(* CODESYS project Door.xml

Project tree, tasks and I/O mapping:
  function block Door [LD]
*)

// Door
FUNCTION_BLOCK Door
// The Door function block monitors the conditions required for locking and unlocking the door.
// The door should remained locked until a bag of ice is ready to be vended.
VAR_INPUT
	Enable:				BOOL;
	DoorClosed: 		BOOL; 				// Inductive prox input to detect the door closed.
	KickerBlocked: 		BOOL; 				// Photoelectric sensor input to detect if a bag is still on the kicker.
	DoorLocked: 		BOOL; 				// Output from the door lock if the lock is successfully locked.
	Unlock: 			BOOL;				// Input from control sequence to unlock when the bag of ice is ready.
	AutoDoorLock:		BOOL;
	IgnoreKicker:		BOOL;
	CheckLockDelay:		TIME;				// Time to wait before checking lock status
END_VAR
VAR_OUTPUT
	Lock: 				BOOL; 				// Output to the door lock.
	DoorLockFault: 		BOOL; 				// Output bit for a fault condition if the door fails to lock.
END_VAR
VAR
	_TimeUnlocked: 		TIME;
	_TimeLocked: 		TIME;
	_CheckLockTimer: 	TON;
END_VAR

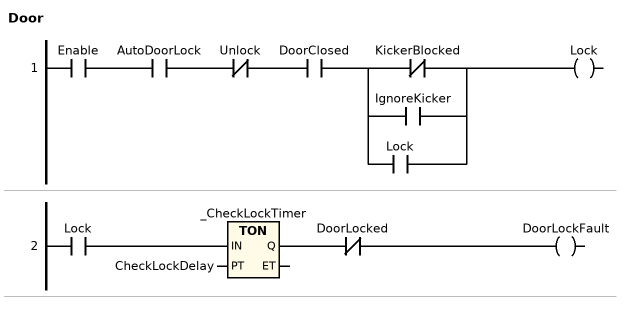
// NETWORK 1
Lock := Enable AND AutoDoorLock AND NOT Unlock AND DoorClosed AND (NOT KickerBlocked OR IgnoreKicker OR Lock);

// NETWORK 2
_CheckLockTimer(IN := Lock, PT := CheckLockDelay); // TON
DoorLockFault := _CheckLockTimer.Q AND NOT DoorLocked;

END_FUNCTION_BLOCK
